TYPE "LBP_typeTMLoad"
TITLE = Tool management / Gestión de herramientas / Werkzeugverwaltung
// User data type for block LBP_TMLoad [DB71] / Tipo de dato de usuario para bloque LBP_TMLoad [DB71] / Anwender-Datentyp für Baustein LBP_TMLoad [DB71]
// stored: IsFailsafeCompliant false
   STRUCT
      IFNo : Array[1..16] of Bool;   // Schnittstelle [Nummer] aktiv / Interface [number] active / Interfaz [número] activa
      Quit : Array[1..16] of Bool;   // Quit-End durchführen / Perform Quit-End / Ejecutar Finalizar confirmación
      TIF : Array[1..16] of Struct
         Loading : Bool;   // Werkzeug wird geladen / Loading the tool / Cargando herramienta
         Unloading : Bool;   // Werkzeug wird entladen / Unloading the tool / Descargando herramienta
         Reloading : Bool;   // Tool wird neu positioniert / Relocating the tool / Reposicionado de herramienta
         Positioning : Bool;   // Magazin wird positioniert / Positioning the magazine / Posicionando almacén
         PosbyProgram : Bool;   // Veranlassung durch CNC-Programm / Initiation by CNC program / Inicio desde programa CNC
         PositioningMT : Bool;   // Multitool wird positioniert / Positioning multitool / Posicionando Multitool
         f0_6 : Bool;   // Reserviert / Reserved / Reservado
         f0_7 : Bool;   // Reserviert / Reserved / Reservado
         PerfStatusError : Bool;   // Negative Quittung / Negative acknowledge / Confirmación negativa
         n1_1 : Bool;   // Reserviert / Reserved / Reservado
         n1_2 : Bool;   // Reserviert / Reserved / Reservado
         n1_3 : Bool;   // Reserviert / Reserved / Reservado
         n1_4 : Bool;   // Reserviert / Reserved / Reservado
         n1_5 : Bool;   // Reserviert / Reserved / Reservado
         n1_6 : Bool;   // Reserviert / Reserved / Reservado
         DataInDB1071 : Bool;   // Multitool-Daten gespeichert in DB1071 / Multitool data stored in DB1071 / Datos Multitool guardados en DB1071
         Channel : Byte;   // Zugeordneter Kanal / Assigned channel / Canal asignado
         TMNo : Byte;   // Werkzeug-Verwaltungsnummer / Tool management number / Número de gestión de herramientas
         reserved1 : DInt;   // Reserviert / Reserved / Reservado
         reserved2 : DInt;   // Reserviert / Reserved / Reservado
         reserved3 : DInt;   // Reserviert / Reserved / Reservado
         LoadIdent : Int;   // Identifikation für Lade-/Entladestation / Identification for loading/unloading station / Identificación para estación de carga/descarga
         LoadNo : Int;   // Nummer der Ladestation / Number of loading station / Número de estación de carga
         SMag : Int;   // Magazin-Nummer (Quelle) für Entladen/Neuladen/Pos. / Magazine number (source) for unloading/reloading/pos. / Número de almacén (origen) para descargar/cargar de nuevo/pos.
         SLoc : Int;   // Platznummer (Quelle) für Entladen/Neuladen/Pos. / Location number (source) for unloading/reloading/pos. / Número de puesto (origen) para descargar/cargar de nuevo/pos.
         TMag : Int;   // Magazin-Nummer (Ziel) für Laden/Neuladen / Magazine number (target) for loading/reloading / Número de almacén (destino) para descargar/cargar de nuevo
         TLoc : Int;   // Platznummer (Ziel) für Laden/Neuladen / Location number (target) for loading/reloading / Número de puesto (destino) para descargar/cargar de nuevo
         WithoutMagMoving : Bool;   // HMI-Daten ohne Magazinbewegung / HMI Data: without magazine moving / Datos HMI sin movimiento de almacén
         Res2 : Byte;   // Reserviert / Reserved / Reservado
      END_STRUCT;
   END_STRUCT;
   // // TIF[2].Loading : Werkzeug wird geladen / Loading the tool / Cargando herramienta
   // // TIF[3].Loading : Werkzeug wird geladen / Loading the tool / Cargando herramienta
   // // TIF[4].Loading : Werkzeug wird geladen / Loading the tool / Cargando herramienta
   // // TIF[5].Loading : Werkzeug wird geladen / Loading the tool / Cargando herramienta
   // // TIF[6].Loading : Werkzeug wird geladen / Loading the tool / Cargando herramienta
   // // TIF[7].Loading : Werkzeug wird geladen / Loading the tool / Cargando herramienta
   // // TIF[8].Loading : Werkzeug wird geladen / Loading the tool / Cargando herramienta
   // // TIF[9].Loading : Werkzeug wird geladen / Loading the tool / Cargando herramienta
   // // TIF[10].Loading : Werkzeug wird geladen / Loading the tool / Cargando herramienta
   // // TIF[11].Loading : Werkzeug wird geladen / Loading the tool / Cargando herramienta
   // // TIF[12].Loading : Werkzeug wird geladen / Loading the tool / Cargando herramienta
   // // TIF[13].Loading : Werkzeug wird geladen / Loading the tool / Cargando herramienta
   // // TIF[14].Loading : Werkzeug wird geladen / Loading the tool / Cargando herramienta
   // // TIF[15].Loading : Werkzeug wird geladen / Loading the tool / Cargando herramienta
   // // TIF[16].Loading : Werkzeug wird geladen / Loading the tool / Cargando herramienta
   // // TIF[2].Unloading : Werkzeug wird entladen / Unloading the tool / Descargando herramienta
   // // TIF[3].Unloading : Werkzeug wird entladen / Unloading the tool / Descargando herramienta
   // // TIF[4].Unloading : Werkzeug wird entladen / Unloading the tool / Descargando herramienta
   // // TIF[5].Unloading : Werkzeug wird entladen / Unloading the tool / Descargando herramienta
   // // TIF[6].Unloading : Werkzeug wird entladen / Unloading the tool / Descargando herramienta
   // // TIF[7].Unloading : Werkzeug wird entladen / Unloading the tool / Descargando herramienta
   // // TIF[8].Unloading : Werkzeug wird entladen / Unloading the tool / Descargando herramienta
   // // TIF[9].Unloading : Werkzeug wird entladen / Unloading the tool / Descargando herramienta
   // // TIF[10].Unloading : Werkzeug wird entladen / Unloading the tool / Descargando herramienta
   // // TIF[11].Unloading : Werkzeug wird entladen / Unloading the tool / Descargando herramienta
   // // TIF[12].Unloading : Werkzeug wird entladen / Unloading the tool / Descargando herramienta
   // // TIF[13].Unloading : Werkzeug wird entladen / Unloading the tool / Descargando herramienta
   // // TIF[14].Unloading : Werkzeug wird entladen / Unloading the tool / Descargando herramienta
   // // TIF[15].Unloading : Werkzeug wird entladen / Unloading the tool / Descargando herramienta
   // // TIF[16].Unloading : Werkzeug wird entladen / Unloading the tool / Descargando herramienta
   // // TIF[2].Reloading : Tool wird neu positioniert / Relocating the tool / Reposicionado de herramienta
   // // TIF[3].Reloading : Tool wird neu positioniert / Relocating the tool / Reposicionado de herramienta
   // // TIF[4].Reloading : Tool wird neu positioniert / Relocating the tool / Reposicionado de herramienta
   // // TIF[5].Reloading : Tool wird neu positioniert / Relocating the tool / Reposicionado de herramienta
   // // TIF[6].Reloading : Tool wird neu positioniert / Relocating the tool / Reposicionado de herramienta
   // // TIF[7].Reloading : Tool wird neu positioniert / Relocating the tool / Reposicionado de herramienta
   // // TIF[8].Reloading : Tool wird neu positioniert / Relocating the tool / Reposicionado de herramienta
   // // TIF[9].Reloading : Tool wird neu positioniert / Relocating the tool / Reposicionado de herramienta
   // // TIF[10].Reloading : Tool wird neu positioniert / Relocating the tool / Reposicionado de herramienta
   // // TIF[11].Reloading : Tool wird neu positioniert / Relocating the tool / Reposicionado de herramienta
   // // TIF[12].Reloading : Tool wird neu positioniert / Relocating the tool / Reposicionado de herramienta
   // // TIF[13].Reloading : Tool wird neu positioniert / Relocating the tool / Reposicionado de herramienta
   // // TIF[14].Reloading : Tool wird neu positioniert / Relocating the tool / Reposicionado de herramienta
   // // TIF[15].Reloading : Tool wird neu positioniert / Relocating the tool / Reposicionado de herramienta
   // // TIF[16].Reloading : Tool wird neu positioniert / Relocating the tool / Reposicionado de herramienta
   // // TIF[2].Positioning : Magazin wird positioniert / Positioning the magazine / Posicionando almacén
   // // TIF[3].Positioning : Magazin wird positioniert / Positioning the magazine / Posicionando almacén
   // // TIF[4].Positioning : Magazin wird positioniert / Positioning the magazine / Posicionando almacén
   // // TIF[5].Positioning : Magazin wird positioniert / Positioning the magazine / Posicionando almacén
   // // TIF[6].Positioning : Magazin wird positioniert / Positioning the magazine / Posicionando almacén
   // // TIF[7].Positioning : Magazin wird positioniert / Positioning the magazine / Posicionando almacén
   // // TIF[8].Positioning : Magazin wird positioniert / Positioning the magazine / Posicionando almacén
   // // TIF[9].Positioning : Magazin wird positioniert / Positioning the magazine / Posicionando almacén
   // // TIF[10].Positioning : Magazin wird positioniert / Positioning the magazine / Posicionando almacén
   // // TIF[11].Positioning : Magazin wird positioniert / Positioning the magazine / Posicionando almacén
   // // TIF[12].Positioning : Magazin wird positioniert / Positioning the magazine / Posicionando almacén
   // // TIF[13].Positioning : Magazin wird positioniert / Positioning the magazine / Posicionando almacén
   // // TIF[14].Positioning : Magazin wird positioniert / Positioning the magazine / Posicionando almacén
   // // TIF[15].Positioning : Magazin wird positioniert / Positioning the magazine / Posicionando almacén
   // // TIF[16].Positioning : Magazin wird positioniert / Positioning the magazine / Posicionando almacén
   // // TIF[2].PosbyProgram : Veranlassung durch CNC-Programm / Initiation by CNC program / Inicio desde programa CNC
   // // TIF[3].PosbyProgram : Veranlassung durch CNC-Programm / Initiation by CNC program / Inicio desde programa CNC
   // // TIF[4].PosbyProgram : Veranlassung durch CNC-Programm / Initiation by CNC program / Inicio desde programa CNC
   // // TIF[5].PosbyProgram : Veranlassung durch CNC-Programm / Initiation by CNC program / Inicio desde programa CNC
   // // TIF[6].PosbyProgram : Veranlassung durch CNC-Programm / Initiation by CNC program / Inicio desde programa CNC
   // // TIF[7].PosbyProgram : Veranlassung durch CNC-Programm / Initiation by CNC program / Inicio desde programa CNC
   // // TIF[8].PosbyProgram : Veranlassung durch CNC-Programm / Initiation by CNC program / Inicio desde programa CNC
   // // TIF[9].PosbyProgram : Veranlassung durch CNC-Programm / Initiation by CNC program / Inicio desde programa CNC
   // // TIF[10].PosbyProgram : Veranlassung durch CNC-Programm / Initiation by CNC program / Inicio desde programa CNC
   // // TIF[11].PosbyProgram : Veranlassung durch CNC-Programm / Initiation by CNC program / Inicio desde programa CNC
   // // TIF[12].PosbyProgram : Veranlassung durch CNC-Programm / Initiation by CNC program / Inicio desde programa CNC
   // // TIF[13].PosbyProgram : Veranlassung durch CNC-Programm / Initiation by CNC program / Inicio desde programa CNC
   // // TIF[14].PosbyProgram : Veranlassung durch CNC-Programm / Initiation by CNC program / Inicio desde programa CNC
   // // TIF[15].PosbyProgram : Veranlassung durch CNC-Programm / Initiation by CNC program / Inicio desde programa CNC
   // // TIF[16].PosbyProgram : Veranlassung durch CNC-Programm / Initiation by CNC program / Inicio desde programa CNC
   // // TIF[2].PositioningMT : Multitool wird positioniert / Positioning multitool / Posicionando Multitool
   // // TIF[3].PositioningMT : Multitool wird positioniert / Positioning multitool / Posicionando Multitool
   // // TIF[4].PositioningMT : Multitool wird positioniert / Positioning multitool / Posicionando Multitool
   // // TIF[5].PositioningMT : Multitool wird positioniert / Positioning multitool / Posicionando Multitool
   // // TIF[6].PositioningMT : Multitool wird positioniert / Positioning multitool / Posicionando Multitool
   // // TIF[7].PositioningMT : Multitool wird positioniert / Positioning multitool / Posicionando Multitool
   // // TIF[8].PositioningMT : Multitool wird positioniert / Positioning multitool / Posicionando Multitool
   // // TIF[9].PositioningMT : Multitool wird positioniert / Positioning multitool / Posicionando Multitool
   // // TIF[10].PositioningMT : Multitool wird positioniert / Positioning multitool / Posicionando Multitool
   // // TIF[11].PositioningMT : Multitool wird positioniert / Positioning multitool / Posicionando Multitool
   // // TIF[12].PositioningMT : Multitool wird positioniert / Positioning multitool / Posicionando Multitool
   // // TIF[13].PositioningMT : Multitool wird positioniert / Positioning multitool / Posicionando Multitool
   // // TIF[14].PositioningMT : Multitool wird positioniert / Positioning multitool / Posicionando Multitool
   // // TIF[15].PositioningMT : Multitool wird positioniert / Positioning multitool / Posicionando Multitool
   // // TIF[16].PositioningMT : Multitool wird positioniert / Positioning multitool / Posicionando Multitool
   // // TIF[2].f0_6 : Reserviert / Reserved / Reservado
   // // TIF[3].f0_6 : Reserviert / Reserved / Reservado
   // // TIF[4].f0_6 : Reserviert / Reserved / Reservado
   // // TIF[5].f0_6 : Reserviert / Reserved / Reservado
   // // TIF[6].f0_6 : Reserviert / Reserved / Reservado
   // // TIF[7].f0_6 : Reserviert / Reserved / Reservado
   // // TIF[8].f0_6 : Reserviert / Reserved / Reservado
   // // TIF[9].f0_6 : Reserviert / Reserved / Reservado
   // // TIF[10].f0_6 : Reserviert / Reserved / Reservado
   // // TIF[11].f0_6 : Reserviert / Reserved / Reservado
   // // TIF[12].f0_6 : Reserviert / Reserved / Reservado
   // // TIF[13].f0_6 : Reserviert / Reserved / Reservado
   // // TIF[14].f0_6 : Reserviert / Reserved / Reservado
   // // TIF[15].f0_6 : Reserviert / Reserved / Reservado
   // // TIF[16].f0_6 : Reserviert / Reserved / Reservado
   // // TIF[2].f0_7 : Reserviert / Reserved / Reservado
   // // TIF[3].f0_7 : Reserviert / Reserved / Reservado
   // // TIF[4].f0_7 : Reserviert / Reserved / Reservado
   // // TIF[5].f0_7 : Reserviert / Reserved / Reservado
   // // TIF[6].f0_7 : Reserviert / Reserved / Reservado
   // // TIF[7].f0_7 : Reserviert / Reserved / Reservado
   // // TIF[8].f0_7 : Reserviert / Reserved / Reservado
   // // TIF[9].f0_7 : Reserviert / Reserved / Reservado
   // // TIF[10].f0_7 : Reserviert / Reserved / Reservado
   // // TIF[11].f0_7 : Reserviert / Reserved / Reservado
   // // TIF[12].f0_7 : Reserviert / Reserved / Reservado
   // // TIF[13].f0_7 : Reserviert / Reserved / Reservado
   // // TIF[14].f0_7 : Reserviert / Reserved / Reservado
   // // TIF[15].f0_7 : Reserviert / Reserved / Reservado
   // // TIF[16].f0_7 : Reserviert / Reserved / Reservado
   // // TIF[2].PerfStatusError : Negative Quittung / Negative acknowledge / Confirmación negativa
   // // TIF[3].PerfStatusError : Negative Quittung / Negative acknowledge / Confirmación negativa
   // // TIF[4].PerfStatusError : Negative Quittung / Negative acknowledge / Confirmación negativa
   // // TIF[5].PerfStatusError : Negative Quittung / Negative acknowledge / Confirmación negativa
   // // TIF[6].PerfStatusError : Negative Quittung / Negative acknowledge / Confirmación negativa
   // // TIF[7].PerfStatusError : Negative Quittung / Negative acknowledge / Confirmación negativa
   // // TIF[8].PerfStatusError : Negative Quittung / Negative acknowledge / Confirmación negativa
   // // TIF[9].PerfStatusError : Negative Quittung / Negative acknowledge / Confirmación negativa
   // // TIF[10].PerfStatusError : Negative Quittung / Negative acknowledge / Confirmación negativa
   // // TIF[11].PerfStatusError : Negative Quittung / Negative acknowledge / Confirmación negativa
   // // TIF[12].PerfStatusError : Negative Quittung / Negative acknowledge / Confirmación negativa
   // // TIF[13].PerfStatusError : Negative Quittung / Negative acknowledge / Confirmación negativa
   // // TIF[14].PerfStatusError : Negative Quittung / Negative acknowledge / Confirmación negativa
   // // TIF[15].PerfStatusError : Negative Quittung / Negative acknowledge / Confirmación negativa
   // // TIF[16].PerfStatusError : Negative Quittung / Negative acknowledge / Confirmación negativa
   // // TIF[2].n1_1 : Reserviert / Reserved / Reservado
   // // TIF[3].n1_1 : Reserviert / Reserved / Reservado
   // // TIF[4].n1_1 : Reserviert / Reserved / Reservado
   // // TIF[5].n1_1 : Reserviert / Reserved / Reservado
   // // TIF[6].n1_1 : Reserviert / Reserved / Reservado
   // // TIF[7].n1_1 : Reserviert / Reserved / Reservado
   // // TIF[8].n1_1 : Reserviert / Reserved / Reservado
   // // TIF[9].n1_1 : Reserviert / Reserved / Reservado
   // // TIF[10].n1_1 : Reserviert / Reserved / Reservado
   // // TIF[11].n1_1 : Reserviert / Reserved / Reservado
   // // TIF[12].n1_1 : Reserviert / Reserved / Reservado
   // // TIF[13].n1_1 : Reserviert / Reserved / Reservado
   // // TIF[14].n1_1 : Reserviert / Reserved / Reservado
   // // TIF[15].n1_1 : Reserviert / Reserved / Reservado
   // // TIF[16].n1_1 : Reserviert / Reserved / Reservado
   // // TIF[2].n1_2 : Reserviert / Reserved / Reservado
   // // TIF[3].n1_2 : Reserviert / Reserved / Reservado
   // // TIF[4].n1_2 : Reserviert / Reserved / Reservado
   // // TIF[5].n1_2 : Reserviert / Reserved / Reservado
   // // TIF[6].n1_2 : Reserviert / Reserved / Reservado
   // // TIF[7].n1_2 : Reserviert / Reserved / Reservado
   // // TIF[8].n1_2 : Reserviert / Reserved / Reservado
   // // TIF[9].n1_2 : Reserviert / Reserved / Reservado
   // // TIF[10].n1_2 : Reserviert / Reserved / Reservado
   // // TIF[11].n1_2 : Reserviert / Reserved / Reservado
   // // TIF[12].n1_2 : Reserviert / Reserved / Reservado
   // // TIF[13].n1_2 : Reserviert / Reserved / Reservado
   // // TIF[14].n1_2 : Reserviert / Reserved / Reservado
   // // TIF[15].n1_2 : Reserviert / Reserved / Reservado
   // // TIF[16].n1_2 : Reserviert / Reserved / Reservado
   // // TIF[2].n1_3 : Reserviert / Reserved / Reservado
   // // TIF[3].n1_3 : Reserviert / Reserved / Reservado
   // // TIF[4].n1_3 : Reserviert / Reserved / Reservado
   // // TIF[5].n1_3 : Reserviert / Reserved / Reservado
   // // TIF[6].n1_3 : Reserviert / Reserved / Reservado
   // // TIF[7].n1_3 : Reserviert / Reserved / Reservado
   // // TIF[8].n1_3 : Reserviert / Reserved / Reservado
   // // TIF[9].n1_3 : Reserviert / Reserved / Reservado
   // // TIF[10].n1_3 : Reserviert / Reserved / Reservado
   // // TIF[11].n1_3 : Reserviert / Reserved / Reservado
   // // TIF[12].n1_3 : Reserviert / Reserved / Reservado
   // // TIF[13].n1_3 : Reserviert / Reserved / Reservado
   // // TIF[14].n1_3 : Reserviert / Reserved / Reservado
   // // TIF[15].n1_3 : Reserviert / Reserved / Reservado
   // // TIF[16].n1_3 : Reserviert / Reserved / Reservado
   // // TIF[2].n1_4 : Reserviert / Reserved / Reservado
   // // TIF[3].n1_4 : Reserviert / Reserved / Reservado
   // // TIF[4].n1_4 : Reserviert / Reserved / Reservado
   // // TIF[5].n1_4 : Reserviert / Reserved / Reservado
   // // TIF[6].n1_4 : Reserviert / Reserved / Reservado
   // // TIF[7].n1_4 : Reserviert / Reserved / Reservado
   // // TIF[8].n1_4 : Reserviert / Reserved / Reservado
   // // TIF[9].n1_4 : Reserviert / Reserved / Reservado
   // // TIF[10].n1_4 : Reserviert / Reserved / Reservado
   // // TIF[11].n1_4 : Reserviert / Reserved / Reservado
   // // TIF[12].n1_4 : Reserviert / Reserved / Reservado
   // // TIF[13].n1_4 : Reserviert / Reserved / Reservado
   // // TIF[14].n1_4 : Reserviert / Reserved / Reservado
   // // TIF[15].n1_4 : Reserviert / Reserved / Reservado
   // // TIF[16].n1_4 : Reserviert / Reserved / Reservado
   // // TIF[2].n1_5 : Reserviert / Reserved / Reservado
   // // TIF[3].n1_5 : Reserviert / Reserved / Reservado
   // // TIF[4].n1_5 : Reserviert / Reserved / Reservado
   // // TIF[5].n1_5 : Reserviert / Reserved / Reservado
   // // TIF[6].n1_5 : Reserviert / Reserved / Reservado
   // // TIF[7].n1_5 : Reserviert / Reserved / Reservado
   // // TIF[8].n1_5 : Reserviert / Reserved / Reservado
   // // TIF[9].n1_5 : Reserviert / Reserved / Reservado
   // // TIF[10].n1_5 : Reserviert / Reserved / Reservado
   // // TIF[11].n1_5 : Reserviert / Reserved / Reservado
   // // TIF[12].n1_5 : Reserviert / Reserved / Reservado
   // // TIF[13].n1_5 : Reserviert / Reserved / Reservado
   // // TIF[14].n1_5 : Reserviert / Reserved / Reservado
   // // TIF[15].n1_5 : Reserviert / Reserved / Reservado
   // // TIF[16].n1_5 : Reserviert / Reserved / Reservado
   // // TIF[2].n1_6 : Reserviert / Reserved / Reservado
   // // TIF[3].n1_6 : Reserviert / Reserved / Reservado
   // // TIF[4].n1_6 : Reserviert / Reserved / Reservado
   // // TIF[5].n1_6 : Reserviert / Reserved / Reservado
   // // TIF[6].n1_6 : Reserviert / Reserved / Reservado
   // // TIF[7].n1_6 : Reserviert / Reserved / Reservado
   // // TIF[8].n1_6 : Reserviert / Reserved / Reservado
   // // TIF[9].n1_6 : Reserviert / Reserved / Reservado
   // // TIF[10].n1_6 : Reserviert / Reserved / Reservado
   // // TIF[11].n1_6 : Reserviert / Reserved / Reservado
   // // TIF[12].n1_6 : Reserviert / Reserved / Reservado
   // // TIF[13].n1_6 : Reserviert / Reserved / Reservado
   // // TIF[14].n1_6 : Reserviert / Reserved / Reservado
   // // TIF[15].n1_6 : Reserviert / Reserved / Reservado
   // // TIF[16].n1_6 : Reserviert / Reserved / Reservado
   // // TIF[2].DataInDB1071 : Multitool-Daten gespeichert in DB1071 / Multitool data stored in DB1071 / Datos Multitool guardados en DB1071
   // // TIF[3].DataInDB1071 : Multitool-Daten gespeichert in DB1071 / Multitool data stored in DB1071 / Datos Multitool guardados en DB1071
   // // TIF[4].DataInDB1071 : Multitool-Daten gespeichert in DB1071 / Multitool data stored in DB1071 / Datos Multitool guardados en DB1071
   // // TIF[5].DataInDB1071 : Multitool-Daten gespeichert in DB1071 / Multitool data stored in DB1071 / Datos Multitool guardados en DB1071
   // // TIF[6].DataInDB1071 : Multitool-Daten gespeichert in DB1071 / Multitool data stored in DB1071 / Datos Multitool guardados en DB1071
   // // TIF[7].DataInDB1071 : Multitool-Daten gespeichert in DB1071 / Multitool data stored in DB1071 / Datos Multitool guardados en DB1071
   // // TIF[8].DataInDB1071 : Multitool-Daten gespeichert in DB1071 / Multitool data stored in DB1071 / Datos Multitool guardados en DB1071
   // // TIF[9].DataInDB1071 : Multitool-Daten gespeichert in DB1071 / Multitool data stored in DB1071 / Datos Multitool guardados en DB1071
   // // TIF[10].DataInDB1071 : Multitool-Daten gespeichert in DB1071 / Multitool data stored in DB1071 / Datos Multitool guardados en DB1071
   // // TIF[11].DataInDB1071 : Multitool-Daten gespeichert in DB1071 / Multitool data stored in DB1071 / Datos Multitool guardados en DB1071
   // // TIF[12].DataInDB1071 : Multitool-Daten gespeichert in DB1071 / Multitool data stored in DB1071 / Datos Multitool guardados en DB1071
   // // TIF[13].DataInDB1071 : Multitool-Daten gespeichert in DB1071 / Multitool data stored in DB1071 / Datos Multitool guardados en DB1071
   // // TIF[14].DataInDB1071 : Multitool-Daten gespeichert in DB1071 / Multitool data stored in DB1071 / Datos Multitool guardados en DB1071
   // // TIF[15].DataInDB1071 : Multitool-Daten gespeichert in DB1071 / Multitool data stored in DB1071 / Datos Multitool guardados en DB1071
   // // TIF[16].DataInDB1071 : Multitool-Daten gespeichert in DB1071 / Multitool data stored in DB1071 / Datos Multitool guardados en DB1071
   // // TIF[2].Channel : Zugeordneter Kanal / Assigned channel / Canal asignado
   // // TIF[3].Channel : Zugeordneter Kanal / Assigned channel / Canal asignado
   // // TIF[4].Channel : Zugeordneter Kanal / Assigned channel / Canal asignado
   // // TIF[5].Channel : Zugeordneter Kanal / Assigned channel / Canal asignado
   // // TIF[6].Channel : Zugeordneter Kanal / Assigned channel / Canal asignado
   // // TIF[7].Channel : Zugeordneter Kanal / Assigned channel / Canal asignado
   // // TIF[8].Channel : Zugeordneter Kanal / Assigned channel / Canal asignado
   // // TIF[9].Channel : Zugeordneter Kanal / Assigned channel / Canal asignado
   // // TIF[10].Channel : Zugeordneter Kanal / Assigned channel / Canal asignado
   // // TIF[11].Channel : Zugeordneter Kanal / Assigned channel / Canal asignado
   // // TIF[12].Channel : Zugeordneter Kanal / Assigned channel / Canal asignado
   // // TIF[13].Channel : Zugeordneter Kanal / Assigned channel / Canal asignado
   // // TIF[14].Channel : Zugeordneter Kanal / Assigned channel / Canal asignado
   // // TIF[15].Channel : Zugeordneter Kanal / Assigned channel / Canal asignado
   // // TIF[16].Channel : Zugeordneter Kanal / Assigned channel / Canal asignado
   // // TIF[2].TMNo : Werkzeug-Verwaltungsnummer / Tool management number / Número de gestión de herramientas
   // // TIF[3].TMNo : Werkzeug-Verwaltungsnummer / Tool management number / Número de gestión de herramientas
   // // TIF[4].TMNo : Werkzeug-Verwaltungsnummer / Tool management number / Número de gestión de herramientas
   // // TIF[5].TMNo : Werkzeug-Verwaltungsnummer / Tool management number / Número de gestión de herramientas
   // // TIF[6].TMNo : Werkzeug-Verwaltungsnummer / Tool management number / Número de gestión de herramientas
   // // TIF[7].TMNo : Werkzeug-Verwaltungsnummer / Tool management number / Número de gestión de herramientas
   // // TIF[8].TMNo : Werkzeug-Verwaltungsnummer / Tool management number / Número de gestión de herramientas
   // // TIF[9].TMNo : Werkzeug-Verwaltungsnummer / Tool management number / Número de gestión de herramientas
   // // TIF[10].TMNo : Werkzeug-Verwaltungsnummer / Tool management number / Número de gestión de herramientas
   // // TIF[11].TMNo : Werkzeug-Verwaltungsnummer / Tool management number / Número de gestión de herramientas
   // // TIF[12].TMNo : Werkzeug-Verwaltungsnummer / Tool management number / Número de gestión de herramientas
   // // TIF[13].TMNo : Werkzeug-Verwaltungsnummer / Tool management number / Número de gestión de herramientas
   // // TIF[14].TMNo : Werkzeug-Verwaltungsnummer / Tool management number / Número de gestión de herramientas
   // // TIF[15].TMNo : Werkzeug-Verwaltungsnummer / Tool management number / Número de gestión de herramientas
   // // TIF[16].TMNo : Werkzeug-Verwaltungsnummer / Tool management number / Número de gestión de herramientas
   // // TIF[2].reserved1 : Reserviert / Reserved / Reservado
   // // TIF[3].reserved1 : Reserviert / Reserved / Reservado
   // // TIF[4].reserved1 : Reserviert / Reserved / Reservado
   // // TIF[5].reserved1 : Reserviert / Reserved / Reservado
   // // TIF[6].reserved1 : Reserviert / Reserved / Reservado
   // // TIF[7].reserved1 : Reserviert / Reserved / Reservado
   // // TIF[8].reserved1 : Reserviert / Reserved / Reservado
   // // TIF[9].reserved1 : Reserviert / Reserved / Reservado
   // // TIF[10].reserved1 : Reserviert / Reserved / Reservado
   // // TIF[11].reserved1 : Reserviert / Reserved / Reservado
   // // TIF[12].reserved1 : Reserviert / Reserved / Reservado
   // // TIF[13].reserved1 : Reserviert / Reserved / Reservado
   // // TIF[14].reserved1 : Reserviert / Reserved / Reservado
   // // TIF[15].reserved1 : Reserviert / Reserved / Reservado
   // // TIF[16].reserved1 : Reserviert / Reserved / Reservado
   // // TIF[2].reserved2 : Reserviert / Reserved / Reservado
   // // TIF[3].reserved2 : Reserviert / Reserved / Reservado
   // // TIF[4].reserved2 : Reserviert / Reserved / Reservado
   // // TIF[5].reserved2 : Reserviert / Reserved / Reservado
   // // TIF[6].reserved2 : Reserviert / Reserved / Reservado
   // // TIF[7].reserved2 : Reserviert / Reserved / Reservado
   // // TIF[8].reserved2 : Reserviert / Reserved / Reservado
   // // TIF[9].reserved2 : Reserviert / Reserved / Reservado
   // // TIF[10].reserved2 : Reserviert / Reserved / Reservado
   // // TIF[11].reserved2 : Reserviert / Reserved / Reservado
   // // TIF[12].reserved2 : Reserviert / Reserved / Reservado
   // // TIF[13].reserved2 : Reserviert / Reserved / Reservado
   // // TIF[14].reserved2 : Reserviert / Reserved / Reservado
   // // TIF[15].reserved2 : Reserviert / Reserved / Reservado
   // // TIF[16].reserved2 : Reserviert / Reserved / Reservado
   // // TIF[2].reserved3 : Reserviert / Reserved / Reservado
   // // TIF[3].reserved3 : Reserviert / Reserved / Reservado
   // // TIF[4].reserved3 : Reserviert / Reserved / Reservado
   // // TIF[5].reserved3 : Reserviert / Reserved / Reservado
   // // TIF[6].reserved3 : Reserviert / Reserved / Reservado
   // // TIF[7].reserved3 : Reserviert / Reserved / Reservado
   // // TIF[8].reserved3 : Reserviert / Reserved / Reservado
   // // TIF[9].reserved3 : Reserviert / Reserved / Reservado
   // // TIF[10].reserved3 : Reserviert / Reserved / Reservado
   // // TIF[11].reserved3 : Reserviert / Reserved / Reservado
   // // TIF[12].reserved3 : Reserviert / Reserved / Reservado
   // // TIF[13].reserved3 : Reserviert / Reserved / Reservado
   // // TIF[14].reserved3 : Reserviert / Reserved / Reservado
   // // TIF[15].reserved3 : Reserviert / Reserved / Reservado
   // // TIF[16].reserved3 : Reserviert / Reserved / Reservado
   // // TIF[2].LoadIdent : Identifikation für Lade-/Entladestation / Identification for loading/unloading station / Identificación para estación de carga/descarga
   // // TIF[3].LoadIdent : Identifikation für Lade-/Entladestation / Identification for loading/unloading station / Identificación para estación de carga/descarga
   // // TIF[4].LoadIdent : Identifikation für Lade-/Entladestation / Identification for loading/unloading station / Identificación para estación de carga/descarga
   // // TIF[5].LoadIdent : Identifikation für Lade-/Entladestation / Identification for loading/unloading station / Identificación para estación de carga/descarga
   // // TIF[6].LoadIdent : Identifikation für Lade-/Entladestation / Identification for loading/unloading station / Identificación para estación de carga/descarga
   // // TIF[7].LoadIdent : Identifikation für Lade-/Entladestation / Identification for loading/unloading station / Identificación para estación de carga/descarga
   // // TIF[8].LoadIdent : Identifikation für Lade-/Entladestation / Identification for loading/unloading station / Identificación para estación de carga/descarga
   // // TIF[9].LoadIdent : Identifikation für Lade-/Entladestation / Identification for loading/unloading station / Identificación para estación de carga/descarga
   // // TIF[10].LoadIdent : Identifikation für Lade-/Entladestation / Identification for loading/unloading station / Identificación para estación de carga/descarga
   // // TIF[11].LoadIdent : Identifikation für Lade-/Entladestation / Identification for loading/unloading station / Identificación para estación de carga/descarga
   // // TIF[12].LoadIdent : Identifikation für Lade-/Entladestation / Identification for loading/unloading station / Identificación para estación de carga/descarga
   // // TIF[13].LoadIdent : Identifikation für Lade-/Entladestation / Identification for loading/unloading station / Identificación para estación de carga/descarga
   // // TIF[14].LoadIdent : Identifikation für Lade-/Entladestation / Identification for loading/unloading station / Identificación para estación de carga/descarga
   // // TIF[15].LoadIdent : Identifikation für Lade-/Entladestation / Identification for loading/unloading station / Identificación para estación de carga/descarga
   // // TIF[16].LoadIdent : Identifikation für Lade-/Entladestation / Identification for loading/unloading station / Identificación para estación de carga/descarga
   // // TIF[2].LoadNo : Nummer der Ladestation / Number of loading station / Número de estación de carga
   // // TIF[3].LoadNo : Nummer der Ladestation / Number of loading station / Número de estación de carga
   // // TIF[4].LoadNo : Nummer der Ladestation / Number of loading station / Número de estación de carga
   // // TIF[5].LoadNo : Nummer der Ladestation / Number of loading station / Número de estación de carga
   // // TIF[6].LoadNo : Nummer der Ladestation / Number of loading station / Número de estación de carga
   // // TIF[7].LoadNo : Nummer der Ladestation / Number of loading station / Número de estación de carga
   // // TIF[8].LoadNo : Nummer der Ladestation / Number of loading station / Número de estación de carga
   // // TIF[9].LoadNo : Nummer der Ladestation / Number of loading station / Número de estación de carga
   // // TIF[10].LoadNo : Nummer der Ladestation / Number of loading station / Número de estación de carga
   // // TIF[11].LoadNo : Nummer der Ladestation / Number of loading station / Número de estación de carga
   // // TIF[12].LoadNo : Nummer der Ladestation / Number of loading station / Número de estación de carga
   // // TIF[13].LoadNo : Nummer der Ladestation / Number of loading station / Número de estación de carga
   // // TIF[14].LoadNo : Nummer der Ladestation / Number of loading station / Número de estación de carga
   // // TIF[15].LoadNo : Nummer der Ladestation / Number of loading station / Número de estación de carga
   // // TIF[16].LoadNo : Nummer der Ladestation / Number of loading station / Número de estación de carga
   // // TIF[2].SMag : Magazin-Nummer (Quelle) für Entladen/Neuladen/Pos. / Magazine number (source) for unloading/reloading/pos. / Número de almacén (origen) para descargar/cargar de nuevo/pos.
   // // TIF[3].SMag : Magazin-Nummer (Quelle) für Entladen/Neuladen/Pos. / Magazine number (source) for unloading/reloading/pos. / Número de almacén (origen) para descargar/cargar de nuevo/pos.
   // // TIF[4].SMag : Magazin-Nummer (Quelle) für Entladen/Neuladen/Pos. / Magazine number (source) for unloading/reloading/pos. / Número de almacén (origen) para descargar/cargar de nuevo/pos.
   // // TIF[5].SMag : Magazin-Nummer (Quelle) für Entladen/Neuladen/Pos. / Magazine number (source) for unloading/reloading/pos. / Número de almacén (origen) para descargar/cargar de nuevo/pos.
   // // TIF[6].SMag : Magazin-Nummer (Quelle) für Entladen/Neuladen/Pos. / Magazine number (source) for unloading/reloading/pos. / Número de almacén (origen) para descargar/cargar de nuevo/pos.
   // // TIF[7].SMag : Magazin-Nummer (Quelle) für Entladen/Neuladen/Pos. / Magazine number (source) for unloading/reloading/pos. / Número de almacén (origen) para descargar/cargar de nuevo/pos.
   // // TIF[8].SMag : Magazin-Nummer (Quelle) für Entladen/Neuladen/Pos. / Magazine number (source) for unloading/reloading/pos. / Número de almacén (origen) para descargar/cargar de nuevo/pos.
   // // TIF[9].SMag : Magazin-Nummer (Quelle) für Entladen/Neuladen/Pos. / Magazine number (source) for unloading/reloading/pos. / Número de almacén (origen) para descargar/cargar de nuevo/pos.
   // // TIF[10].SMag : Magazin-Nummer (Quelle) für Entladen/Neuladen/Pos. / Magazine number (source) for unloading/reloading/pos. / Número de almacén (origen) para descargar/cargar de nuevo/pos.
   // // TIF[11].SMag : Magazin-Nummer (Quelle) für Entladen/Neuladen/Pos. / Magazine number (source) for unloading/reloading/pos. / Número de almacén (origen) para descargar/cargar de nuevo/pos.
   // // TIF[12].SMag : Magazin-Nummer (Quelle) für Entladen/Neuladen/Pos. / Magazine number (source) for unloading/reloading/pos. / Número de almacén (origen) para descargar/cargar de nuevo/pos.
   // // TIF[13].SMag : Magazin-Nummer (Quelle) für Entladen/Neuladen/Pos. / Magazine number (source) for unloading/reloading/pos. / Número de almacén (origen) para descargar/cargar de nuevo/pos.
   // // TIF[14].SMag : Magazin-Nummer (Quelle) für Entladen/Neuladen/Pos. / Magazine number (source) for unloading/reloading/pos. / Número de almacén (origen) para descargar/cargar de nuevo/pos.
   // // TIF[15].SMag : Magazin-Nummer (Quelle) für Entladen/Neuladen/Pos. / Magazine number (source) for unloading/reloading/pos. / Número de almacén (origen) para descargar/cargar de nuevo/pos.
   // // TIF[16].SMag : Magazin-Nummer (Quelle) für Entladen/Neuladen/Pos. / Magazine number (source) for unloading/reloading/pos. / Número de almacén (origen) para descargar/cargar de nuevo/pos.
   // // TIF[2].SLoc : Platznummer (Quelle) für Entladen/Neuladen/Pos. / Location number (source) for unloading/reloading/pos. / Número de puesto (origen) para descargar/cargar de nuevo/pos.
   // // TIF[3].SLoc : Platznummer (Quelle) für Entladen/Neuladen/Pos. / Location number (source) for unloading/reloading/pos. / Número de puesto (origen) para descargar/cargar de nuevo/pos.
   // // TIF[4].SLoc : Platznummer (Quelle) für Entladen/Neuladen/Pos. / Location number (source) for unloading/reloading/pos. / Número de puesto (origen) para descargar/cargar de nuevo/pos.
   // // TIF[5].SLoc : Platznummer (Quelle) für Entladen/Neuladen/Pos. / Location number (source) for unloading/reloading/pos. / Número de puesto (origen) para descargar/cargar de nuevo/pos.
   // // TIF[6].SLoc : Platznummer (Quelle) für Entladen/Neuladen/Pos. / Location number (source) for unloading/reloading/pos. / Número de puesto (origen) para descargar/cargar de nuevo/pos.
   // // TIF[7].SLoc : Platznummer (Quelle) für Entladen/Neuladen/Pos. / Location number (source) for unloading/reloading/pos. / Número de puesto (origen) para descargar/cargar de nuevo/pos.
   // // TIF[8].SLoc : Platznummer (Quelle) für Entladen/Neuladen/Pos. / Location number (source) for unloading/reloading/pos. / Número de puesto (origen) para descargar/cargar de nuevo/pos.
   // // TIF[9].SLoc : Platznummer (Quelle) für Entladen/Neuladen/Pos. / Location number (source) for unloading/reloading/pos. / Número de puesto (origen) para descargar/cargar de nuevo/pos.
   // // TIF[10].SLoc : Platznummer (Quelle) für Entladen/Neuladen/Pos. / Location number (source) for unloading/reloading/pos. / Número de puesto (origen) para descargar/cargar de nuevo/pos.
   // // TIF[11].SLoc : Platznummer (Quelle) für Entladen/Neuladen/Pos. / Location number (source) for unloading/reloading/pos. / Número de puesto (origen) para descargar/cargar de nuevo/pos.
   // // TIF[12].SLoc : Platznummer (Quelle) für Entladen/Neuladen/Pos. / Location number (source) for unloading/reloading/pos. / Número de puesto (origen) para descargar/cargar de nuevo/pos.
   // // TIF[13].SLoc : Platznummer (Quelle) für Entladen/Neuladen/Pos. / Location number (source) for unloading/reloading/pos. / Número de puesto (origen) para descargar/cargar de nuevo/pos.
   // // TIF[14].SLoc : Platznummer (Quelle) für Entladen/Neuladen/Pos. / Location number (source) for unloading/reloading/pos. / Número de puesto (origen) para descargar/cargar de nuevo/pos.
   // // TIF[15].SLoc : Platznummer (Quelle) für Entladen/Neuladen/Pos. / Location number (source) for unloading/reloading/pos. / Número de puesto (origen) para descargar/cargar de nuevo/pos.
   // // TIF[16].SLoc : Platznummer (Quelle) für Entladen/Neuladen/Pos. / Location number (source) for unloading/reloading/pos. / Número de puesto (origen) para descargar/cargar de nuevo/pos.
   // // TIF[2].TMag : Magazin-Nummer (Ziel) für Laden/Neuladen / Magazine number (target) for loading/reloading / Número de almacén (destino) para descargar/cargar de nuevo
   // // TIF[3].TMag : Magazin-Nummer (Ziel) für Laden/Neuladen / Magazine number (target) for loading/reloading / Número de almacén (destino) para descargar/cargar de nuevo
   // // TIF[4].TMag : Magazin-Nummer (Ziel) für Laden/Neuladen / Magazine number (target) for loading/reloading / Número de almacén (destino) para descargar/cargar de nuevo
   // // TIF[5].TMag : Magazin-Nummer (Ziel) für Laden/Neuladen / Magazine number (target) for loading/reloading / Número de almacén (destino) para descargar/cargar de nuevo
   // // TIF[6].TMag : Magazin-Nummer (Ziel) für Laden/Neuladen / Magazine number (target) for loading/reloading / Número de almacén (destino) para descargar/cargar de nuevo
   // // TIF[7].TMag : Magazin-Nummer (Ziel) für Laden/Neuladen / Magazine number (target) for loading/reloading / Número de almacén (destino) para descargar/cargar de nuevo
   // // TIF[8].TMag : Magazin-Nummer (Ziel) für Laden/Neuladen / Magazine number (target) for loading/reloading / Número de almacén (destino) para descargar/cargar de nuevo
   // // TIF[9].TMag : Magazin-Nummer (Ziel) für Laden/Neuladen / Magazine number (target) for loading/reloading / Número de almacén (destino) para descargar/cargar de nuevo
   // // TIF[10].TMag : Magazin-Nummer (Ziel) für Laden/Neuladen / Magazine number (target) for loading/reloading / Número de almacén (destino) para descargar/cargar de nuevo
   // // TIF[11].TMag : Magazin-Nummer (Ziel) für Laden/Neuladen / Magazine number (target) for loading/reloading / Número de almacén (destino) para descargar/cargar de nuevo
   // // TIF[12].TMag : Magazin-Nummer (Ziel) für Laden/Neuladen / Magazine number (target) for loading/reloading / Número de almacén (destino) para descargar/cargar de nuevo
   // // TIF[13].TMag : Magazin-Nummer (Ziel) für Laden/Neuladen / Magazine number (target) for loading/reloading / Número de almacén (destino) para descargar/cargar de nuevo
   // // TIF[14].TMag : Magazin-Nummer (Ziel) für Laden/Neuladen / Magazine number (target) for loading/reloading / Número de almacén (destino) para descargar/cargar de nuevo
   // // TIF[15].TMag : Magazin-Nummer (Ziel) für Laden/Neuladen / Magazine number (target) for loading/reloading / Número de almacén (destino) para descargar/cargar de nuevo
   // // TIF[16].TMag : Magazin-Nummer (Ziel) für Laden/Neuladen / Magazine number (target) for loading/reloading / Número de almacén (destino) para descargar/cargar de nuevo
   // // TIF[2].TLoc : Platznummer (Ziel) für Laden/Neuladen / Location number (target) for loading/reloading / Número de puesto (destino) para descargar/cargar de nuevo
   // // TIF[3].TLoc : Platznummer (Ziel) für Laden/Neuladen / Location number (target) for loading/reloading / Número de puesto (destino) para descargar/cargar de nuevo
   // // TIF[4].TLoc : Platznummer (Ziel) für Laden/Neuladen / Location number (target) for loading/reloading / Número de puesto (destino) para descargar/cargar de nuevo
   // // TIF[5].TLoc : Platznummer (Ziel) für Laden/Neuladen / Location number (target) for loading/reloading / Número de puesto (destino) para descargar/cargar de nuevo
   // // TIF[6].TLoc : Platznummer (Ziel) für Laden/Neuladen / Location number (target) for loading/reloading / Número de puesto (destino) para descargar/cargar de nuevo
   // // TIF[7].TLoc : Platznummer (Ziel) für Laden/Neuladen / Location number (target) for loading/reloading / Número de puesto (destino) para descargar/cargar de nuevo
   // // TIF[8].TLoc : Platznummer (Ziel) für Laden/Neuladen / Location number (target) for loading/reloading / Número de puesto (destino) para descargar/cargar de nuevo
   // // TIF[9].TLoc : Platznummer (Ziel) für Laden/Neuladen / Location number (target) for loading/reloading / Número de puesto (destino) para descargar/cargar de nuevo
   // // TIF[10].TLoc : Platznummer (Ziel) für Laden/Neuladen / Location number (target) for loading/reloading / Número de puesto (destino) para descargar/cargar de nuevo
   // // TIF[11].TLoc : Platznummer (Ziel) für Laden/Neuladen / Location number (target) for loading/reloading / Número de puesto (destino) para descargar/cargar de nuevo
   // // TIF[12].TLoc : Platznummer (Ziel) für Laden/Neuladen / Location number (target) for loading/reloading / Número de puesto (destino) para descargar/cargar de nuevo
   // // TIF[13].TLoc : Platznummer (Ziel) für Laden/Neuladen / Location number (target) for loading/reloading / Número de puesto (destino) para descargar/cargar de nuevo
   // // TIF[14].TLoc : Platznummer (Ziel) für Laden/Neuladen / Location number (target) for loading/reloading / Número de puesto (destino) para descargar/cargar de nuevo
   // // TIF[15].TLoc : Platznummer (Ziel) für Laden/Neuladen / Location number (target) for loading/reloading / Número de puesto (destino) para descargar/cargar de nuevo
   // // TIF[16].TLoc : Platznummer (Ziel) für Laden/Neuladen / Location number (target) for loading/reloading / Número de puesto (destino) para descargar/cargar de nuevo
   // // TIF[2].WithoutMagMoving : HMI-Daten ohne Magazinbewegung / HMI Data: without magazine moving / Datos HMI sin movimiento de almacén
   // // TIF[3].WithoutMagMoving : HMI-Daten ohne Magazinbewegung / HMI Data: without magazine moving / Datos HMI sin movimiento de almacén
   // // TIF[4].WithoutMagMoving : HMI-Daten ohne Magazinbewegung / HMI Data: without magazine moving / Datos HMI sin movimiento de almacén
   // // TIF[5].WithoutMagMoving : HMI-Daten ohne Magazinbewegung / HMI Data: without magazine moving / Datos HMI sin movimiento de almacén
   // // TIF[6].WithoutMagMoving : HMI-Daten ohne Magazinbewegung / HMI Data: without magazine moving / Datos HMI sin movimiento de almacén
   // // TIF[7].WithoutMagMoving : HMI-Daten ohne Magazinbewegung / HMI Data: without magazine moving / Datos HMI sin movimiento de almacén
   // // TIF[8].WithoutMagMoving : HMI-Daten ohne Magazinbewegung / HMI Data: without magazine moving / Datos HMI sin movimiento de almacén
   // // TIF[9].WithoutMagMoving : HMI-Daten ohne Magazinbewegung / HMI Data: without magazine moving / Datos HMI sin movimiento de almacén
   // // TIF[10].WithoutMagMoving : HMI-Daten ohne Magazinbewegung / HMI Data: without magazine moving / Datos HMI sin movimiento de almacén
   // // TIF[11].WithoutMagMoving : HMI-Daten ohne Magazinbewegung / HMI Data: without magazine moving / Datos HMI sin movimiento de almacén
   // // TIF[12].WithoutMagMoving : HMI-Daten ohne Magazinbewegung / HMI Data: without magazine moving / Datos HMI sin movimiento de almacén
   // // TIF[13].WithoutMagMoving : HMI-Daten ohne Magazinbewegung / HMI Data: without magazine moving / Datos HMI sin movimiento de almacén
   // // TIF[14].WithoutMagMoving : HMI-Daten ohne Magazinbewegung / HMI Data: without magazine moving / Datos HMI sin movimiento de almacén
   // // TIF[15].WithoutMagMoving : HMI-Daten ohne Magazinbewegung / HMI Data: without magazine moving / Datos HMI sin movimiento de almacén
   // // TIF[16].WithoutMagMoving : HMI-Daten ohne Magazinbewegung / HMI Data: without magazine moving / Datos HMI sin movimiento de almacén
   // // TIF[2].Res2 : Reserviert / Reserved / Reservado
   // // TIF[3].Res2 : Reserviert / Reserved / Reservado
   // // TIF[4].Res2 : Reserviert / Reserved / Reservado
   // // TIF[5].Res2 : Reserviert / Reserved / Reservado
   // // TIF[6].Res2 : Reserviert / Reserved / Reservado
   // // TIF[7].Res2 : Reserviert / Reserved / Reservado
   // // TIF[8].Res2 : Reserviert / Reserved / Reservado
   // // TIF[9].Res2 : Reserviert / Reserved / Reservado
   // // TIF[10].Res2 : Reserviert / Reserved / Reservado
   // // TIF[11].Res2 : Reserviert / Reserved / Reservado
   // // TIF[12].Res2 : Reserviert / Reserved / Reservado
   // // TIF[13].Res2 : Reserviert / Reserved / Reservado
   // // TIF[14].Res2 : Reserviert / Reserved / Reservado
   // // TIF[15].Res2 : Reserviert / Reserved / Reservado
   // // TIF[16].Res2 : Reserviert / Reserved / Reservado
END_TYPE

TYPE "LBP_typeTMLoadMT"
TITLE = Tool management / Gestión de herramientas / Werkzeugverwaltung
// User data type for block LBP_TMLoadMT [DB1071] / Tipo de dato de usuario para bloque LBP_TMLoadMT [DB1071] / Anwender-Datentyp für Baustein LBP_TMLoadMT [DB1071]
// stored: IsFailsafeCompliant false
   STRUCT
      MTIF : Array[1..16] of Struct
         DistanceCoding : Int;   // Art der Entfernungscodierung ($TC_MTP_KD) / Type of distance coding ($TC_MTP_KD) / Tipo de codificación de distancia ($TC_MTP_KD)
         Places : Int;   // Anzahl der Plätze des Multitools / Number of locations of the multitool / Número de puestos de Multitool
         Distance : Real;   // Entfernung des Multitool-Platzes / Multitool location distance / Distancia a puesto Multitool
         MTNo : Int;   // Interne WZ-Nummer des Multitools / Internal T number of the multitool / Número de herramienta interno de Multitool
         PlaceNo : Int;   // Platznummer im Multitool, auf die das System positioniert / Location number within the multitool to which the system positions / Número de puesto de Multitool en el que posiciona el sistema
         Toolholder : Int;   // Spindel- oder Werkzeughalter-Nummer / Spindle or toolholder number / Número de cabezal o de portaherramientas
         reserved : Array[1..3] of Int;   // Reserviert / Reserved / Reservado
      END_STRUCT;
   END_STRUCT;
   // // MTIF[2].DistanceCoding : Art der Entfernungscodierung ($TC_MTP_KD) / Type of distance coding ($TC_MTP_KD) / Tipo de codificación de distancia ($TC_MTP_KD)
   // // MTIF[3].DistanceCoding : Art der Entfernungscodierung ($TC_MTP_KD) / Type of distance coding ($TC_MTP_KD) / Tipo de codificación de distancia ($TC_MTP_KD)
   // // MTIF[4].DistanceCoding : Art der Entfernungscodierung ($TC_MTP_KD) / Type of distance coding ($TC_MTP_KD) / Tipo de codificación de distancia ($TC_MTP_KD)
   // // MTIF[5].DistanceCoding : Art der Entfernungscodierung ($TC_MTP_KD) / Type of distance coding ($TC_MTP_KD) / Tipo de codificación de distancia ($TC_MTP_KD)
   // // MTIF[6].DistanceCoding : Art der Entfernungscodierung ($TC_MTP_KD) / Type of distance coding ($TC_MTP_KD) / Tipo de codificación de distancia ($TC_MTP_KD)
   // // MTIF[7].DistanceCoding : Art der Entfernungscodierung ($TC_MTP_KD) / Type of distance coding ($TC_MTP_KD) / Tipo de codificación de distancia ($TC_MTP_KD)
   // // MTIF[8].DistanceCoding : Art der Entfernungscodierung ($TC_MTP_KD) / Type of distance coding ($TC_MTP_KD) / Tipo de codificación de distancia ($TC_MTP_KD)
   // // MTIF[9].DistanceCoding : Art der Entfernungscodierung ($TC_MTP_KD) / Type of distance coding ($TC_MTP_KD) / Tipo de codificación de distancia ($TC_MTP_KD)
   // // MTIF[10].DistanceCoding : Art der Entfernungscodierung ($TC_MTP_KD) / Type of distance coding ($TC_MTP_KD) / Tipo de codificación de distancia ($TC_MTP_KD)
   // // MTIF[11].DistanceCoding : Art der Entfernungscodierung ($TC_MTP_KD) / Type of distance coding ($TC_MTP_KD) / Tipo de codificación de distancia ($TC_MTP_KD)
   // // MTIF[12].DistanceCoding : Art der Entfernungscodierung ($TC_MTP_KD) / Type of distance coding ($TC_MTP_KD) / Tipo de codificación de distancia ($TC_MTP_KD)
   // // MTIF[13].DistanceCoding : Art der Entfernungscodierung ($TC_MTP_KD) / Type of distance coding ($TC_MTP_KD) / Tipo de codificación de distancia ($TC_MTP_KD)
   // // MTIF[14].DistanceCoding : Art der Entfernungscodierung ($TC_MTP_KD) / Type of distance coding ($TC_MTP_KD) / Tipo de codificación de distancia ($TC_MTP_KD)
   // // MTIF[15].DistanceCoding : Art der Entfernungscodierung ($TC_MTP_KD) / Type of distance coding ($TC_MTP_KD) / Tipo de codificación de distancia ($TC_MTP_KD)
   // // MTIF[16].DistanceCoding : Art der Entfernungscodierung ($TC_MTP_KD) / Type of distance coding ($TC_MTP_KD) / Tipo de codificación de distancia ($TC_MTP_KD)
   // // MTIF[2].Places : Anzahl der Plätze des Multitools / Number of locations of the multitool / Número de puestos de Multitool
   // // MTIF[3].Places : Anzahl der Plätze des Multitools / Number of locations of the multitool / Número de puestos de Multitool
   // // MTIF[4].Places : Anzahl der Plätze des Multitools / Number of locations of the multitool / Número de puestos de Multitool
   // // MTIF[5].Places : Anzahl der Plätze des Multitools / Number of locations of the multitool / Número de puestos de Multitool
   // // MTIF[6].Places : Anzahl der Plätze des Multitools / Number of locations of the multitool / Número de puestos de Multitool
   // // MTIF[7].Places : Anzahl der Plätze des Multitools / Number of locations of the multitool / Número de puestos de Multitool
   // // MTIF[8].Places : Anzahl der Plätze des Multitools / Number of locations of the multitool / Número de puestos de Multitool
   // // MTIF[9].Places : Anzahl der Plätze des Multitools / Number of locations of the multitool / Número de puestos de Multitool
   // // MTIF[10].Places : Anzahl der Plätze des Multitools / Number of locations of the multitool / Número de puestos de Multitool
   // // MTIF[11].Places : Anzahl der Plätze des Multitools / Number of locations of the multitool / Número de puestos de Multitool
   // // MTIF[12].Places : Anzahl der Plätze des Multitools / Number of locations of the multitool / Número de puestos de Multitool
   // // MTIF[13].Places : Anzahl der Plätze des Multitools / Number of locations of the multitool / Número de puestos de Multitool
   // // MTIF[14].Places : Anzahl der Plätze des Multitools / Number of locations of the multitool / Número de puestos de Multitool
   // // MTIF[15].Places : Anzahl der Plätze des Multitools / Number of locations of the multitool / Número de puestos de Multitool
   // // MTIF[16].Places : Anzahl der Plätze des Multitools / Number of locations of the multitool / Número de puestos de Multitool
   // // MTIF[2].Distance : Entfernung des Multitool-Platzes / Multitool location distance / Distancia a puesto Multitool
   // // MTIF[3].Distance : Entfernung des Multitool-Platzes / Multitool location distance / Distancia a puesto Multitool
   // // MTIF[4].Distance : Entfernung des Multitool-Platzes / Multitool location distance / Distancia a puesto Multitool
   // // MTIF[5].Distance : Entfernung des Multitool-Platzes / Multitool location distance / Distancia a puesto Multitool
   // // MTIF[6].Distance : Entfernung des Multitool-Platzes / Multitool location distance / Distancia a puesto Multitool
   // // MTIF[7].Distance : Entfernung des Multitool-Platzes / Multitool location distance / Distancia a puesto Multitool
   // // MTIF[8].Distance : Entfernung des Multitool-Platzes / Multitool location distance / Distancia a puesto Multitool
   // // MTIF[9].Distance : Entfernung des Multitool-Platzes / Multitool location distance / Distancia a puesto Multitool
   // // MTIF[10].Distance : Entfernung des Multitool-Platzes / Multitool location distance / Distancia a puesto Multitool
   // // MTIF[11].Distance : Entfernung des Multitool-Platzes / Multitool location distance / Distancia a puesto Multitool
   // // MTIF[12].Distance : Entfernung des Multitool-Platzes / Multitool location distance / Distancia a puesto Multitool
   // // MTIF[13].Distance : Entfernung des Multitool-Platzes / Multitool location distance / Distancia a puesto Multitool
   // // MTIF[14].Distance : Entfernung des Multitool-Platzes / Multitool location distance / Distancia a puesto Multitool
   // // MTIF[15].Distance : Entfernung des Multitool-Platzes / Multitool location distance / Distancia a puesto Multitool
   // // MTIF[16].Distance : Entfernung des Multitool-Platzes / Multitool location distance / Distancia a puesto Multitool
   // // MTIF[2].MTNo : Interne WZ-Nummer des Multitools / Internal T number of the multitool / Número de herramienta interno de Multitool
   // // MTIF[3].MTNo : Interne WZ-Nummer des Multitools / Internal T number of the multitool / Número de herramienta interno de Multitool
   // // MTIF[4].MTNo : Interne WZ-Nummer des Multitools / Internal T number of the multitool / Número de herramienta interno de Multitool
   // // MTIF[5].MTNo : Interne WZ-Nummer des Multitools / Internal T number of the multitool / Número de herramienta interno de Multitool
   // // MTIF[6].MTNo : Interne WZ-Nummer des Multitools / Internal T number of the multitool / Número de herramienta interno de Multitool
   // // MTIF[7].MTNo : Interne WZ-Nummer des Multitools / Internal T number of the multitool / Número de herramienta interno de Multitool
   // // MTIF[8].MTNo : Interne WZ-Nummer des Multitools / Internal T number of the multitool / Número de herramienta interno de Multitool
   // // MTIF[9].MTNo : Interne WZ-Nummer des Multitools / Internal T number of the multitool / Número de herramienta interno de Multitool
   // // MTIF[10].MTNo : Interne WZ-Nummer des Multitools / Internal T number of the multitool / Número de herramienta interno de Multitool
   // // MTIF[11].MTNo : Interne WZ-Nummer des Multitools / Internal T number of the multitool / Número de herramienta interno de Multitool
   // // MTIF[12].MTNo : Interne WZ-Nummer des Multitools / Internal T number of the multitool / Número de herramienta interno de Multitool
   // // MTIF[13].MTNo : Interne WZ-Nummer des Multitools / Internal T number of the multitool / Número de herramienta interno de Multitool
   // // MTIF[14].MTNo : Interne WZ-Nummer des Multitools / Internal T number of the multitool / Número de herramienta interno de Multitool
   // // MTIF[15].MTNo : Interne WZ-Nummer des Multitools / Internal T number of the multitool / Número de herramienta interno de Multitool
   // // MTIF[16].MTNo : Interne WZ-Nummer des Multitools / Internal T number of the multitool / Número de herramienta interno de Multitool
   // // MTIF[2].PlaceNo : Platznummer im Multitool, auf die das System positioniert / Location number within the multitool to which the system positions / Número de puesto de Multitool en el que posiciona el sistema
   // // MTIF[3].PlaceNo : Platznummer im Multitool, auf die das System positioniert / Location number within the multitool to which the system positions / Número de puesto de Multitool en el que posiciona el sistema
   // // MTIF[4].PlaceNo : Platznummer im Multitool, auf die das System positioniert / Location number within the multitool to which the system positions / Número de puesto de Multitool en el que posiciona el sistema
   // // MTIF[5].PlaceNo : Platznummer im Multitool, auf die das System positioniert / Location number within the multitool to which the system positions / Número de puesto de Multitool en el que posiciona el sistema
   // // MTIF[6].PlaceNo : Platznummer im Multitool, auf die das System positioniert / Location number within the multitool to which the system positions / Número de puesto de Multitool en el que posiciona el sistema
   // // MTIF[7].PlaceNo : Platznummer im Multitool, auf die das System positioniert / Location number within the multitool to which the system positions / Número de puesto de Multitool en el que posiciona el sistema
   // // MTIF[8].PlaceNo : Platznummer im Multitool, auf die das System positioniert / Location number within the multitool to which the system positions / Número de puesto de Multitool en el que posiciona el sistema
   // // MTIF[9].PlaceNo : Platznummer im Multitool, auf die das System positioniert / Location number within the multitool to which the system positions / Número de puesto de Multitool en el que posiciona el sistema
   // // MTIF[10].PlaceNo : Platznummer im Multitool, auf die das System positioniert / Location number within the multitool to which the system positions / Número de puesto de Multitool en el que posiciona el sistema
   // // MTIF[11].PlaceNo : Platznummer im Multitool, auf die das System positioniert / Location number within the multitool to which the system positions / Número de puesto de Multitool en el que posiciona el sistema
   // // MTIF[12].PlaceNo : Platznummer im Multitool, auf die das System positioniert / Location number within the multitool to which the system positions / Número de puesto de Multitool en el que posiciona el sistema
   // // MTIF[13].PlaceNo : Platznummer im Multitool, auf die das System positioniert / Location number within the multitool to which the system positions / Número de puesto de Multitool en el que posiciona el sistema
   // // MTIF[14].PlaceNo : Platznummer im Multitool, auf die das System positioniert / Location number within the multitool to which the system positions / Número de puesto de Multitool en el que posiciona el sistema
   // // MTIF[15].PlaceNo : Platznummer im Multitool, auf die das System positioniert / Location number within the multitool to which the system positions / Número de puesto de Multitool en el que posiciona el sistema
   // // MTIF[16].PlaceNo : Platznummer im Multitool, auf die das System positioniert / Location number within the multitool to which the system positions / Número de puesto de Multitool en el que posiciona el sistema
   // // MTIF[2].Toolholder : Spindel- oder Werkzeughalter-Nummer / Spindle or toolholder number / Número de cabezal o de portaherramientas
   // // MTIF[3].Toolholder : Spindel- oder Werkzeughalter-Nummer / Spindle or toolholder number / Número de cabezal o de portaherramientas
   // // MTIF[4].Toolholder : Spindel- oder Werkzeughalter-Nummer / Spindle or toolholder number / Número de cabezal o de portaherramientas
   // // MTIF[5].Toolholder : Spindel- oder Werkzeughalter-Nummer / Spindle or toolholder number / Número de cabezal o de portaherramientas
   // // MTIF[6].Toolholder : Spindel- oder Werkzeughalter-Nummer / Spindle or toolholder number / Número de cabezal o de portaherramientas
   // // MTIF[7].Toolholder : Spindel- oder Werkzeughalter-Nummer / Spindle or toolholder number / Número de cabezal o de portaherramientas
   // // MTIF[8].Toolholder : Spindel- oder Werkzeughalter-Nummer / Spindle or toolholder number / Número de cabezal o de portaherramientas
   // // MTIF[9].Toolholder : Spindel- oder Werkzeughalter-Nummer / Spindle or toolholder number / Número de cabezal o de portaherramientas
   // // MTIF[10].Toolholder : Spindel- oder Werkzeughalter-Nummer / Spindle or toolholder number / Número de cabezal o de portaherramientas
   // // MTIF[11].Toolholder : Spindel- oder Werkzeughalter-Nummer / Spindle or toolholder number / Número de cabezal o de portaherramientas
   // // MTIF[12].Toolholder : Spindel- oder Werkzeughalter-Nummer / Spindle or toolholder number / Número de cabezal o de portaherramientas
   // // MTIF[13].Toolholder : Spindel- oder Werkzeughalter-Nummer / Spindle or toolholder number / Número de cabezal o de portaherramientas
   // // MTIF[14].Toolholder : Spindel- oder Werkzeughalter-Nummer / Spindle or toolholder number / Número de cabezal o de portaherramientas
   // // MTIF[15].Toolholder : Spindel- oder Werkzeughalter-Nummer / Spindle or toolholder number / Número de cabezal o de portaherramientas
   // // MTIF[16].Toolholder : Spindel- oder Werkzeughalter-Nummer / Spindle or toolholder number / Número de cabezal o de portaherramientas
   // // MTIF[2].reserved : Reserviert / Reserved / Reservado
   // // MTIF[3].reserved : Reserviert / Reserved / Reservado
   // // MTIF[4].reserved : Reserviert / Reserved / Reservado
   // // MTIF[5].reserved : Reserviert / Reserved / Reservado
   // // MTIF[6].reserved : Reserviert / Reserved / Reservado
   // // MTIF[7].reserved : Reserviert / Reserved / Reservado
   // // MTIF[8].reserved : Reserviert / Reserved / Reservado
   // // MTIF[9].reserved : Reserviert / Reserved / Reservado
   // // MTIF[10].reserved : Reserviert / Reserved / Reservado
   // // MTIF[11].reserved : Reserviert / Reserved / Reservado
   // // MTIF[12].reserved : Reserviert / Reserved / Reservado
   // // MTIF[13].reserved : Reserviert / Reserved / Reservado
   // // MTIF[14].reserved : Reserviert / Reserved / Reservado
   // // MTIF[15].reserved : Reserviert / Reserved / Reservado
   // // MTIF[16].reserved : Reserviert / Reserved / Reservado
END_TYPE

